(* PLC project main, Beckhoff Automation GmbH TwinCAT PLC Control 3.5.13.21 *)
(* stored: creationDateTime 2022-06-05T16:15:56.4832631, modificationDateTime 2022-06-05T16:15:56.4852631 *)

PROGRAM MAIN
VAR
	ModuleSeperationSensors 		AT%I*		: BYTE := 0;			// 0000_0dmu
	ModuleSeperationActuators		AT%Q*		: BYTE := 0;			// 0000_00rc
	
	sensUp, sensMiddle, sensDown				: BOOL;
	
	sigCreate, sigRemove				: BOOL;
	actUpOpen, actUpClose				: BOOL;
	actDownOpen, actDownClose 			: BOOL;
	
	moduleSeperation		: FB_Separator;
	seperationEnable, seperationExecute	: BOOL;
END_VAR

            // Converting Inputs
sensUp := BYTE_TO_BOOL(ModuleSeperationSensors AND 2#0000_0001);
sensMiddle := BYTE_TO_BOOL(ModuleSeperationSensors AND 2#0000_0010);
sensDown := BYTE_TO_BOOL(ModuleSeperationSensors AND 2#0000_0100);


// Instance calls
moduleSeperation(
	bEnable:= seperationEnable, 
	bExecute:= seperationExecute, 
	bErrorReset:= , 
	bSensor1:= sensDown, 
	bSensor2:= sensMiddle, 
	bSensor3:= sensUp, 
	bR1AKT1=> actUpClose, 
	bR2AKT1=> actUpOpen, 
	bR1AKT2=> actDownOpen, 
	bR2AKT2=> actDownClose, 
	bNoBottle=> , bWrongBottle=> , eStatus=> );


// Converting Outputs
ModuleSeperationActuators := 0;
ModuleSeperationActuators := BOOL_TO_BYTE(sigCreate) OR ModuleSeperationActuators;
ModuleSeperationActuators := SHL(BOOL_TO_BYTE(sigRemove),1) OR ModuleSeperationActuators;

ModuleSeperationActuators := SHL(BOOL_TO_BYTE(actUpOpen),7) OR ModuleSeperationActuators;
ModuleSeperationActuators := SHL(BOOL_TO_BYTE(actUpClose),6) OR ModuleSeperationActuators;
ModuleSeperationActuators := SHL(BOOL_TO_BYTE(actDownOpen),5) OR ModuleSeperationActuators;
ModuleSeperationActuators := SHL(BOOL_TO_BYTE(actDownClose),4) OR ModuleSeperationActuators;

          
END_PROGRAM
